FUNCTION_BLOCK TIMER
  {SET_ATTRIBUTE(OpcUa, DEVICE.SENSOR)}
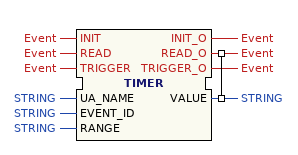
  EVENT_INPUT
    INIT;
    READ;
    TRIGGER;
  END_EVENT
  EVENT_OUTPUT
    INIT_O;
    READ_O WITH VALUE;
    TRIGGER_O;
  END_EVENT
  VAR_INPUT
    UA_NAME : STRING; {SET_ATTRIBUTE(OpcUa, Constant)}
    EVENT_ID : STRING; {SET_ATTRIBUTE(OpcUa, Constant)}
    RANGE : STRING; {SET_ATTRIBUTE(OpcUa, Constant)}
  END_VAR
  VAR_OUTPUT
    VALUE : STRING; {SET_ATTRIBUTE(OpcUa, Variable)}
  END_VAR
END_FUNCTION_BLOCK
